INTERFACE I_NodePrototypes

METHOD PUBLIC Accept
VAR_INPUT
	Visitor : I_NodePrototypeVisitor;
END_VAR
END_METHOD

PROPERTY PUBLIC HasNodePrototypes : BOOL
GET
END_GET
END_PROPERTY

END_INTERFACE

(* stored: Version 1.1.0.1, ProductVersion 3.1.4024.12
   Itf I_NodePrototypes: Id {db51c4b5-809b-4c54-95d5-5fa08c92fe8e}
   Method Accept: Id {20048756-eb31-4de1-bd66-cd1ead8d69a0}
   Property HasNodePrototypes: Id {26e6d624-d752-06f3-2b7f-863472e96820}
   Get Get: Id {23727720-c27c-0a22-104a-393a041d9e2d} *)
